TYPE Alm_AlarmHistoryType :
STRUCT
  	EventMessage:            	WSTRING;
	EventId:					INT;
   	EventTime:               	DT;
END_STRUCT
END_TYPE

(* stored: Version 1.1.0.1, ProductVersion 3.1.4024.12
   DUT Alm_AlarmHistoryType: Id {e001ec5a-2023-4ebc-8eb0-69ba1ddb39ac} *)
